FUNCTION_BLOCK ABSTRACT Xts IMPLEMENTS I_Cyclic, I_Initialisable, I_XTS, I_Object
VAR
	MyName : STRING;
	_MyXts : INT;
	_XtsEnabled : BOOL;
	_XPU : I_TcIoXtsProcessingUnit;
	_MoverArray : ARRAY[0..MaxMovers] OF I_XtsMover;
	_XtsIoEnvVar : I_XtsIoEnvVar;
	ICollisionGroup : I_CollisionGroup;
	_MyXtsHardware : I_XtsHardware;
	XtsHwState : XtsSystemInitialisation;
	EnableSequence : XtsEnableSequence;
	DisableSequence : XtsDisableSequence;	
	Initialised : BOOL;
	EnabledTrigger : R_TRIG;
	DisabledTrigger : R_TRIG;
	_registeredNumberOfMovers: INT;
	DetectedMoverCount : UDINT;
END_VAR
VAR CONSTANT
	MaxMovers : INT := 255;
END_VAR

{analysis -2}

METHOD PUBLIC Cycle : HRESULT
VAR
	EnableResult : HRESULT;
	DisableResult : HRESULT;
	GrpStopResult : HRESULT;
	CollisionResult : HRESULT;
END_VAR
IF Initialised THEN	
	EnableResult := EnableSequence.Cycle();
	DisableResult := DisableSequence.Cycle();
	EnabledTrigger(CLK := EnableSequence.Done);
	DisabledTrigger(CLK := DisableSequence.Done);
	IF EnabledTrigger.Q THEN
		_XtsEnabled := TRUE;
	END_IF
	IF DisabledTrigger.Q THEN
		_XtsEnabled := false;
	END_IF
	IF EnableResult = E_FAIL OR
		DisableResult = E_FAIL OR
		GrpStopResult = E_FAIL OR
		CollisionResult = E_FAIL THEN
		Cycle := E_FAIL;
	END_IF
END_IF
END_METHOD

METHOD DisableXTS : BOOL
VAR_INPUT
END_VAR
IF _XtsEnabled THEN
	DisableXTS := SUCCEEDED(DisableSequence.Disable());
END_IF
END_METHOD

METHOD EnableXTS : BOOL
VAR_INPUT
END_VAR
IF NOT _XtsEnabled THEN
	EnableXts := SUCCEEDED(EnableSequence.Enable());
END_IF
END_METHOD

PROPERTY ExpectedNumberOfParts : int
GET
ExpectedNumberOfParts := _MyXtsHardware.ExpectedNumberOfParts;
END_GET
SET
_MyXtsHardware.ExpectedNumberOfParts := ExpectedNumberOfParts;
END_SET
END_PROPERTY

PROPERTY ExpectedNumberOfTracks : int
GET
ExpectedNumberOfTracks := _MyXtsHardware.ExpectedNumberOfTracks;
END_GET
SET
_MyXtsHardware.ExpectedNumberOfTracks := ExpectedNumberOfTracks;
END_SET
END_PROPERTY

//FB_Init is always available implicitly and it is used primarily for initialization.
//The return value is not evaluated. For a specific influence, you can also declare the
//methods explicitly and provide additional code there with the standard initialization
//code. You can evaluate the return value.
METHOD FB_Init: BOOL
VAR_INPUT
    bInitRetains: BOOL; // TRUE: the retain variables are initialized (reset warm / reset cold)
    bInCopyCode: BOOL;  // TRUE: the instance will be copied to the copy code afterward (online change)   
	MyXtsIoEnvVar : I_XtsIoEnvVar;
	MyXtsHardware : I_XtsHardware;
	MyCAGroup : I_CollisionGroup;
END_VAR
_XtsIoEnvVar := MyXtsIoEnvVar;
_MyXtsHardware := MyXtsHardware;
ICollisionGroup := MyCAGroup;
EnableSequence.MyCollisionGroup := ICollisionGroup;
DisableSequence.MyCollisionGroup := ICollisionGroup;
END_METHOD

METHOD HasError : BOOL
VAR_INPUT
END_VAR
HasError := ICollisionGroup.HasError();
END_METHOD

METHOD Initialise : HRESULT
VAR
	i : INT;
END_VAR
Initialise := -1;
CASE XtsHwState OF
	XtsSystemInitialisation.Init:
		IF _XtsIoEnvVar.IsInitialised() THEN
			_XPU := _XtsIoEnvVar.GetXPUInterface(_MyXts);
			_MyXtsHardware.MyXpu := _XPU;
			XtsHwState := XtsSystemInitialisation.PassGroupReference;
		END_IF
		
	XtsSystemInitialisation.PassGroupReference:
		ICollisionGroup.CAGroupXtsIoEnvInterface := _XtsIoEnvVar.GetCaGroupInterface(_MyXts);
		XtsHwState := XtsSystemInitialisation.InitialiseHardware;
	
	XtsSystemInitialisation.InitialiseHardware:
		IF _MyXtsHardware.IsInitialised() THEN
			MyName := _MyXtsHardware.MyName;
			XtsHwState := XtsSystemInitialisation.SetDetection;
		END_IF
	
	XtsSystemInitialisation.SetDetection:
		IF SUCCEEDED(_MyXtsHardware.SetTrackForDetection(1)) THEN
			XtsHwState := XtsSystemInitialisation.Redetect;
		END_IF
		
	XtsSystemInitialisation.Redetect:
		IF SUCCEEDED(_MyXtsHardware.TriggerRedetection()) THEN
			XtsHwState := XtsSystemInitialisation.MoversValid;
		END_IF
		
	XtsSystemInitialisation.MoversValid:
		IF _MyXtsHardware.AreAllMoversValid() THEN
			XtsHwState := XtsSystemInitialisation.AllMoversFound;
		END_IF
	
	XtsSystemInitialisation.AllMoversFound:
		IF _MyXtsHardware.AreExpectedMoversFound() THEN
			DetectedMoverCount := _MyXtsHardware.getNumberMoversDetected();
			XtsHwState := XtsSystemInitialisation.XTSMode;
		END_IF
		
	XtsSystemInitialisation.XTSMode:
		IF _MyXtsHardware.IsInSim() THEN
			XtsHwState := XtsSystemInitialisation.MoverIdDetection;
		ELSE
			XtsHwState := XtsSystemInitialisation.CheckModuleVoltages;
		END_IF
		
	XtsSystemInitialisation.CheckModuleVoltages:
		IF _MyXtsHardware.Is24VdcOK() = 2 AND _MyXtsHardware.Is48VdcOK() = 2 THEN
			XtsHwState := XtsSystemInitialisation.MoverIdDetection;
		END_IF
	
	XtsSystemInitialisation.MoverIdDetection:
		IF _MyXtsHardware.IsIDDetectionStandard() OR SUCCEEDED(_MyXtsHardware.TriggerMoverID()) THEN
			XtsHwState := XtsSystemInitialisation.HWReady;
		END_IF
	
	XtsSystemInitialisation.HWReady:
		Initialise := 0;
		Initialised := TRUE;	
END_CASE
END_METHOD

METHOD IsInitialised : BOOL
IsInitialised := Initialised;
END_METHOD

METHOD IsXtsIdle : BOOL
VAR_INPUT
END_VAR
IsXtsIdle := DisableSequence.Done;
END_METHOD

METHOD IsXtsReady : BOOL
VAR_INPUT
END_VAR
IsXtsReady := _XtsEnabled;
END_METHOD

METHOD PUBLIC Abstract MoverHomeSequence : BOOL
VAR_INPUT
END_VAR
END_METHOD

PROPERTY MyXts : INT
GET
MyXts := _MyXtsHardware.MyXts;
END_GET
SET
_MyXtsHardware.MyXts := _MyXts := MyXts;
END_SET
END_PROPERTY

METHOD RegisterMovers : HRESULT
VAR_INPUT
	MyMover : I_XtsMover;
END_VAR
VAR
	i : UINT;
	MoverRegistered: BOOL;
END_VAR
IF MyMover = 0 THEN
	RegisterMovers := -1;
	RETURN;
END_IF
IF NOT Initialised THEN
	RegisterMovers := -2;
	RETURN;
END_IF
IF _registeredNumberOfMovers >= MaxMovers THEN
	RegisterMovers := -3;
	RETURN;
END_IF
FOR i := 0 TO (_registeredNumberOfMovers - 1) DO
	IF _MoverArray[i] = MyMover THEN
		MoverRegistered := TRUE;
		EXIT;
	END_IF
END_FOR
IF MoverRegistered THEN
	RegisterMovers := -4;
	RETURN;
END_IF

_MoverArray[_registeredNumberOfMovers] := MyMover;
_registeredNumberOfMovers := _registeredNumberOfMovers + 1;
EnableSequence.RegisterMovers(MyMover);
DisableSequence.RegisterMovers(MyMover);
FOR i := 1 TO _MyXtsHardware.DetectedNumberOfTracks DO
	MyMover.RegisterTracks(Track := _MyXtsHardware.GetTrackByNumber(i));
END_FOR
FOR i := 1 TO TO_UINT(_XPU.GetDetectedMoverCount()) DO
	IF MyMover.AxisRef.NcToPlc.AxisId = _XPU.MoverTcIo(i).GetAxisId() THEN
		MyMover.MoverXtsIoEnvInterface := _XPU.MoverTcIo(i);
	END_IF
END_FOR
END_METHOD

METHOD RegisterWithParent
VAR_INPUT
	Runner	: I_HostObjects;
END_VAR
Runner.RegisterCyclic(THIS^);
Runner.RegisterInitialisable(THIS^);
END_METHOD

METHOD Reset : BOOL
VAR_INPUT
END_VAR
Reset := SUCCEEDED(ICollisionGroup.Reset());
_MyXtsHardware.ResetParts();
END_METHOD

METHOD StopXts : BOOL
VAR_INPUT
END_VAR
StopXTS := ICollisionGroup.GroupStop();
END_METHOD

END_FUNCTION_BLOCK

(* stored: Version 1.1.0.1
   POU Xts: Id {4538c683-94fc-49a1-b5ad-30ffec5e4eff}, SpecialFunc None
   Folder Operations: Id {0e8598c4-3d58-4c14-a12f-6fd3f3ea02bf}
   Folder Settings: Id {cec05bdb-9232-4b5d-b91e-848bd7bc55d9}
   Folder Status: Id {c34f5481-c408-4671-a299-9c4a6e31956c}
   Method Cycle: Id {da42838e-fb00-40a5-96f4-b787aa883566}
   Method DisableXTS: Id {e2a85e5a-c7bf-481d-be4f-81acebc29fb7}
   Method EnableXTS: Id {e800781e-1435-4747-9cb4-9b9fab34ca22}
   Property ExpectedNumberOfParts: Id {33632734-2180-4c77-982d-f6997ead5bb5}
   Get Get: Id {ec285ff9-810a-46b0-8941-68dcdc1ab79d}
   Set Set: Id {4cb5fde4-6845-43ef-b95e-df4929829b0c}
   Property ExpectedNumberOfTracks: Id {6b69c4c6-afe3-46d9-bc08-86224f82f24a}
   Get Get: Id {cab0d03f-ccb1-4d2e-adb6-3d697ceee44c}
   Set Set: Id {b24fc04c-e333-4935-bdff-3eff5a7d9932}
   Method FB_Init: Id {d6ce6c85-5c43-4276-b07f-92a2e669b228}
   Method HasError: Id {deaa9733-0676-46c6-9e2e-c283006fe443}
   Method Initialise: Id {3c52ae7d-89c5-4979-a1bd-5023a279947c}
   Method IsInitialised: Id {ffca4056-5f8a-485d-b64d-57c6377addfd}
   Method IsXtsIdle: Id {98f4e7e8-94b6-4461-9a7b-2bd1c0aafde4}
   Method IsXtsReady: Id {73e2c3f0-1b32-45c2-a8cc-fbf01ac18258}
   Method MoverHomeSequence: Id {5c2deb91-ebd0-4a93-99ec-6a6bbbd5e076}
   Property MyXts: Id {b982f888-fcea-49f3-8b85-76339b257fce}
   Get Get: Id {7260ae55-6d72-4286-9779-c205f4bf658b}
   Set Set: Id {f9bbe24a-eac8-4b47-a949-a650212b0818}
   Method RegisterMovers: Id {a3bbc877-121f-4130-8916-a04d2ba4dd9d}
   Method RegisterWithParent: Id {5a27c335-0022-4ddf-98ff-1436953bbdbd}
   Method Reset: Id {f4cda3e0-308c-460d-87ee-c1616441d1b6}
   Method StopXts: Id {4b648283-f5f4-4d47-a58f-be53e519365d} *)
